ABB RobotStudio station: CV_2_HM.rspag

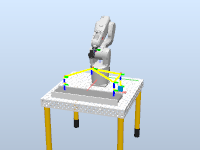
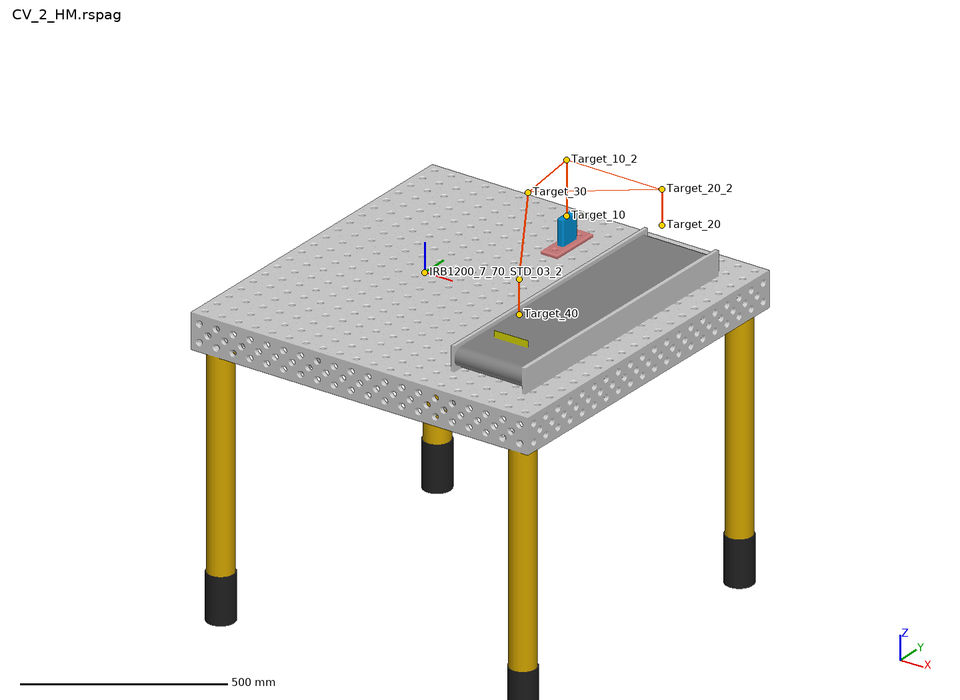
[picture v1: parts stored in the station drawn from their meshes, with robot base, taught points and paths (robot models come from the ABB library and are not in the file)]
--- station ---
Station Solution9 (saved by RobotStudio 21.4.9700.0)
Controller Controller1, task T_ROB1: task frame (RAPID world) sits at (0, 0.8, -98.1) mm in the station
Controller Controller1
  mechanical unit ROB_1: IRB1200_7_70_STD_03_2, 6 joints, base frame (0, 0, 0) mm
Layout (positions relative to the parent item):
  - Workspace [part] at (-401.98, -347.06, -251) mm, size 1010.8 x 1010.8 x 830.4 mm
  - Conveyor [part] at (-401.98, -347.06, -251) mm, size 228.6 x 802.4 x 70.3 mm
  - Object [part] at (-401.98, -347.06, -251) mm, size 20.5 x 60.1 x 75 mm
  - Object_Holder [part] at (-401.98, -347.06, -251) mm, size 51.6 x 150.5 x 10.1 mm
  - Object_Conv_1 [part] at (-120, -350, -196) mm, size 20.5 x 60.1 x 75 mm
  - Object_Sync [part] at (-290, 190, -490) mm, rotated rx 90 ry 0 rz 0 deg, size 20.5 x 60.1 x 75 mm
  - Object_Conv_2 [part] at (-120, -950, -196) mm, size 20.5 x 60.1 x 75 mm
  - IRB1200_7_70_STD_03_2 [mechanism, from Robots\IRB1200_7_70_STD_03.rslib] at (0, 0.8, -98.1) mm; joint values [-0.0452, -0.5689, 1.0507, 0.0672, 0.4271, -0.0968] (rad or m)
  - MyTool [mechanism, from Training Objects\myTool.rslib] at (192.3, -5.62, 405.84) mm, rotated rx -180 ry 38 rz -180 deg
  - PlaneSensor [smart component, from Components\PlaneSensor.rslib] at (46.6, 0, -27.44) mm
      properties: Origin=[0.477982 -0.314586 -0.0004]; Axis1=[0 0 0.02]; Axis2=[-0.1 0 0]; SensedPart=(none)
    - _sensorPart_ [part], size 100 x 0 x 20 mm
  - LinearMover [smart component, from Components\LinearMover.rslib]
      properties: Object=Object; Direction=[0 -0.001 0]; Speed=0.1; Reference=Global; ReferenceObject=(none)
  - Detacher [smart component, from Components\Detacher.rslib]
      properties: Child=Object; KeepPosition=true
  - Attacher [smart component, from Components\Attacher.rslib]
      properties: Parent=MyTool; Flange=0; Child=Object; Mount=false; Offset=[0 0 0]; Orientation=[0 0 0]
  - LogicGate [smart component, from Components\LogicGate.rslib]
      properties: Operator=AND; Delay=0
  - LogicGate_2 [smart component, from Components\LogicGate.rslib]
      properties: Operator=NOT; Delay=0
  - Positioner [smart component, from Components\Positioner.rslib]
      properties: Object=Object; Position=[-0.401984 -0.34706 -0.251]; Orientation=[0 0 0]; Reference=Global; ReferenceObject=(none)
Attachment: MyTool is attached to IRB1200_7_70_STD_03_2 / Link6
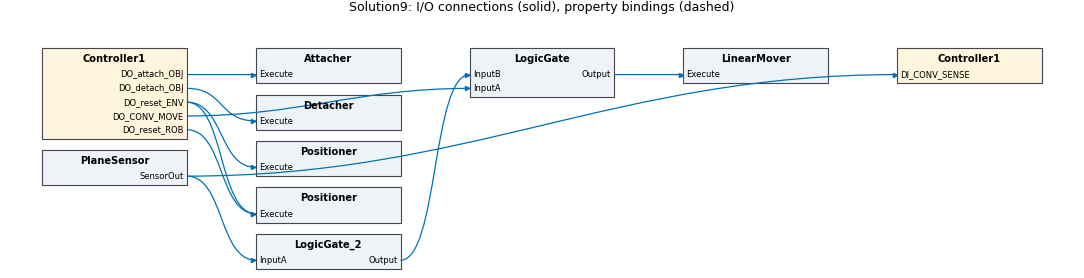
Station logic (signal -> signal, property => property):
  Controller1.DO_attach_OBJ -> Attacher.Execute
  Controller1.DO_detach_OBJ -> Detacher.Execute
  Controller1.DO_reset_ENV -> Positioner.Execute
  PlaneSensor.SensorOut -> Controller1.DI_CONV_SENSE
  LogicGate_2.Output -> LogicGate.InputB
  LogicGate.Output -> LinearMover.Execute
  PlaneSensor.SensorOut -> LogicGate_2.InputA
  Controller1.DO_CONV_MOVE -> LogicGate.InputA
  Controller1.DO_reset_ROB -> Positioner_2.Execute
  Controller1.DO_reset_ENV -> Positioner.Execute

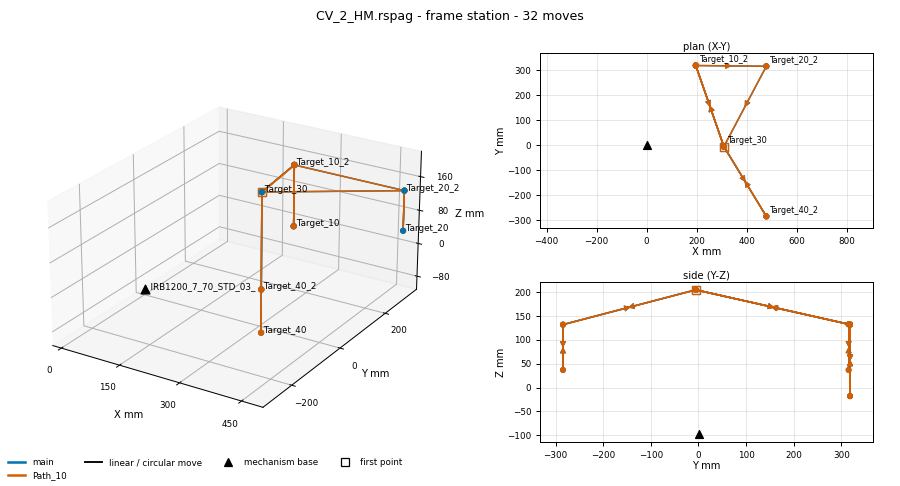
[picture p0: tool path of CV_2_HM.rspag in frame station, 32 of 32 moves have a stored position in this frame; points joined in program order, loops and branches not executed]
--- Backups/Controller1/RAPID/TASK1/PROGMOD/CalibData.mod ---
MODULE CalibData
    PERS tooldata MyTool:=[TRUE,[[31.792631019,0,229.638935148],[0.945518576,0,0.325568154,0]],[1,[0,0,1],[1,0,0,0],0,0,0]];
ENDMODULE

--- Backups/Controller1/RAPID/TASK1/PROGMOD/Module1.mod ---
MODULE Module1
    CONST robtarget Target_30:=[[308.631,-6.416,303.41],[0,0,1,0],[0,0,0,0],[9E+09,9E+09,9E+09,9E+09,9E+09,9E+09]];
    CONST robtarget Target_10_2:=[[196.326,317.543,230.570229267],[0,0,1,0],[0,0,0,0],[9E+09,9E+09,9E+09,9E+09,9E+09,9E+09]];
    CONST robtarget Target_10:=[[196.326,317.543,80.109],[0,0,1,0],[0,-1,1,0],[9E+09,9E+09,9E+09,9E+09,9E+09,9E+09]];
    CONST robtarget Target_20_2:=[[478.311,314.602,230.990771674],[0,0,1,0],[0,0,0,0],[9E+09,9E+09,9E+09,9E+09,9E+09,9E+09]];
    CONST robtarget Target_20:=[[478.311,314.602,135.109],[0,0,1,0],[0,-1,1,0],[9E+09,9E+09,9E+09,9E+09,9E+09,9E+09]];
    CONST robtarget Target_40_2:=[[478.311,-285.398,230.371836045],[0,0,1,0],[-1,0,-2,0],[9E+09,9E+09,9E+09,9E+09,9E+09,9E+09]];
    CONST robtarget Target_40:=[[478.311,-285.398,135.109],[0,0,1,0],[-1,0,-2,0],[9E+09,9E+09,9E+09,9E+09,9E+09,9E+09]];

    !VAR num actual_state;

    PROC main()
        !TEST actual_state
            !CASE 0:
                PulseDO DO_reset_ENV;
                PulseDO DO_detach_OBJ;
                SetDO DO_CONV_MOVE, 0;

                MoveL Target_30,v150,fine,MyTool\WObj:=wobj0;
                MoveL Target_10_2,v150,fine,MyTool\WObj:=wobj0;
                !actual_state := 1;
            !CASE 1:
                !PaP 1
                MoveL Target_10,v150,fine,MyTool\WObj:=wobj0;
                WaitTime 0.1;
                PulseDO DO_attach_OBJ;
                WaitTime 0.1;
                MoveL Target_10_2,v150,fine,MyTool\WObj:=wobj0;
                MoveL Target_20_2,v150,fine,MyTool\WObj:=wobj0;
                MoveL Target_20,v150,fine,MyTool\WObj:=wobj0;
                WaitTime 0.1;
                PulseDO DO_detach_OBJ;
                WaitTime 0.1;
                MoveL Target_20_2,v150,fine,MyTool\WObj:=wobj0;
                !actual_state := 2;
            !CASE 2:
                SetDo DO_CONV_MOVE, 1;
                MoveL Target_30,v150,fine,MyTool\WObj:=wobj0;
                WaitDI DI_CONV_SENSE, 1;
                !actual_state := 3;
            !CASE 3:
                !empty
                IF DI_CONV_SENSE = 1 THEN
                    SetDO DO_CONV_MOVE, 0;
                    !actual_state := 4;
                ENDIF
            !CASE 4:
                !PaP 2
                MoveL Target_40_2,v150,fine,MyTool\WObj:=wobj0;
                MoveL Target_40,v150,fine,MyTool\WObj:=wobj0;
                WaitTime 0.1;
                PulseDO DO_attach_OBJ;
                WaitTime 0.1;
                MoveL Target_40_2,v150,fine,MyTool\WObj:=wobj0;
                MoveL Target_30,v150,fine,MyTool\WObj:=wobj0;
                MoveL Target_10_2,v150,fine,MyTool\WObj:=wobj0;
                MoveL Target_10,v150,fine,MyTool\WObj:=wobj0;
                WaitTime 0.1;
                PulseDO DO_detach_OBJ;
                WaitTime 0.1;
                MoveL Target_10_2,v150,fine,MyTool\WObj:=wobj0;
                MoveL Target_30,v150,fine,MyTool\WObj:=wobj0;
                !actual_state := 10;

            !CASE 10:
                !empty
        !ENDTEST
    ENDPROC



    PROC Path_10()
        MoveL Target_30,v150,fine,MyTool\WObj:=wobj0;
        MoveL Target_10_2,v150,fine,MyTool\WObj:=wobj0;
        MoveL Target_10,v150,fine,MyTool\WObj:=wobj0;
        MoveL Target_10_2,v150,fine,MyTool\WObj:=wobj0;
        MoveL Target_20_2,v150,fine,MyTool\WObj:=wobj0;
        MoveL Target_20,v150,fine,MyTool\WObj:=wobj0;
        MoveL Target_20_2,v150,fine,MyTool\WObj:=wobj0;
        MoveL Target_30,v150,fine,MyTool\WObj:=wobj0;
        MoveL Target_40_2,v150,fine,MyTool\WObj:=wobj0;
        MoveL Target_40,v150,fine,MyTool\WObj:=wobj0;
        MoveL Target_40_2,v150,fine,MyTool\WObj:=wobj0;
        MoveL Target_30,v150,fine,MyTool\WObj:=wobj0;
        MoveL Target_10_2,v150,fine,MyTool\WObj:=wobj0;
        MoveL Target_10,v150,fine,MyTool\WObj:=wobj0;
        MoveL Target_10_2,v150,fine,MyTool\WObj:=wobj0;
        MoveL Target_30,v150,fine,MyTool\WObj:=wobj0;
    ENDPROC
ENDMODULE

--- Backups/Controller1/SYSPAR/EIO.cfg ---
EIO:CFG_1.0:6:1::
#
EIO_SIGNAL:

      -Name "DO_attach_OBJ" -SignalType "DO"

      -Name "DO_detach_OBJ" -SignalType "DO"

      -Name "DO_reset_ENV" -SignalType "DO"

      -Name "DO_CONV_MOVE" -SignalType "DO"

      -Name "DI_CONV_SENSE" -SignalType "DI"

      -Name "DO_reset_ROB" -SignalType "DO"
